// TIA Portal project "2022.10.20_FB_Auto-Hand视觉分拣急停" (V17)
// Vorlageprojekt für das Buch mit Zielsystem S7-1200

(* hardware
DEVICE "S7-1200-Station_1"  S7-1200 Station
   slot 0: "Baugruppenträger_0"  Rack  V1.0
   slot 1: "PLC_1"  CPU 1214C DC/DC/Rly  6ES7 214-1HG40-0XB0  V4.5
DEVICE "HMI_1"  KTP700 Basic PN
   slot 0: "HMI_1"  KTP700 Basic PN  6AV2 123-2GB03-0AX0  17.0.0.0
   slot 1: "HMI_RT_1"  KTP700 Basic PN  6AV2 123-2GB03-0AX0  17.0.0.0
   slot 5: "HMI_1.IE_CP_1"  PROFINET Interface  17.0.0.0
      slot 1: "PROFINET Interface_1"  PROFINET Interface
         slot 1: "Port_1"  Port
*)

// ===== PLC "PLC_1"  CPU 1214C DC/DC/Rly =====

VAR_GLOBAL   // PLC tag table "Standard-Variablentabelle"
   "复位按钮" AT %I0.2 : Bool;
   "System_Byte" AT %MB1 : Byte;
   "FirstScan" AT %M1.0 : Bool;
   "DiagStatusUpdate" AT %M1.1 : Bool;
   "AlwaysTRUE" AT %M1.2 : Bool;
   "AlwaysFALSE" AT %M1.3 : Bool;
   "Clock_Byte" AT %MB0 : Byte;
   "Clock_10Hz" AT %M0.0 : Bool;
   "Clock_5Hz" AT %M0.1 : Bool;
   "Clock_2.5Hz" AT %M0.2 : Bool;
   "Clock_2Hz" AT %M0.3 : Bool;
   "Clock_1.25Hz" AT %M0.4 : Bool;
   "Clock_1Hz" AT %M0.5 : Bool;
   "Clock_0.625Hz" AT %M0.6 : Bool;
   "Clock_0.5Hz" AT %M0.7 : Bool;
END_VAR

VAR_GLOBAL   // PLC tag table "XML 中的变量表_1"
   "启动按钮" AT %I0.0 : Bool;
   "停止按钮" AT %I0.1 : Bool;
   "复位信号" AT %Q0.2 : Bool;
   "急停" AT %I0.3 : Bool;
   "左电传感器" AT %I0.5 : Bool;
   "后电传感器" AT %I0.7 : Bool;
   "手动模式" AT %I1.0 : Bool;
   "自动模式" AT %I1.1 : Bool;
   "启动指示灯" AT %Q0.0 : Bool;
   "停止指示灯" AT %Q0.1 : Bool;
   "送料带" AT %Q0.3 : Bool;
   "直行电机" AT %Q0.4 : Bool;
   "左换向" AT %Q0.5 : Bool;
   "右换向" AT %Q0.6 : Bool;
   "后1带—原料" AT %Q0.7 : Bool;
   "右1带—基座" AT %Q1.0 : Bool;
   "左1带_产品盖" AT %Q1.1 : Bool;
   "出料台" AT %Q1.2 : Bool;
   "挡板" AT %Q1.3 : Bool;
   "视觉相机" AT %ID30 : DWord;
   "右电传感器" AT %I0.6 : Bool;
END_VAR

DATA_BLOCK "主程序DB"   // DB1
{ S7_Optimized_Access := 'TRUE' }
VERSION : 0.1
   VAR
      核心分拣区程序步 : Int;
      启动按钮 : Bool;
      停止按钮 : Bool;
      复位按钮 : Bool;
      急停按钮 : Bool := true;
      "手/自动切换" : Bool;
      中间变量1 : Bool;
      中间变量2 : Bool;
      中间变量3 : Bool;
      中间变量4 : Bool;
      中间变量5 : Bool;
      运行模式 : Int;
   END_VAR
BEGIN
END_DATA_BLOCK

// folder: 01核心分拣区

DATA_BLOCK "视觉核心分拣区FB块_DB"   // DB2
{ S7_Optimized_Access := 'TRUE' }
VERSION : 0.1
// stored: InstanceOfName 视觉核心分拣区FB块
"视觉核心分拣区FB块"
BEGIN
END_DATA_BLOCK

// folder: 02自动运行模式

DATA_BLOCK "自动运行_DB_1"   // DB7
{ S7_Optimized_Access := 'TRUE' }
VERSION : 0.1
// stored: InstanceOfName 自动运行
"自动运行"
BEGIN
END_DATA_BLOCK

// folder: 03手动运行模式

DATA_BLOCK "手动运行_DB"   // DB4
{ S7_Optimized_Access := 'TRUE' }
VERSION : 0.1
// stored: InstanceOfName 手动运行
"手动运行"
BEGIN
END_DATA_BLOCK

DATA_BLOCK "视觉核心分拣区FB块_DB_1"   // DB5
{ S7_Optimized_Access := 'TRUE' }
VERSION : 0.1
// stored: InstanceOfName 视觉核心分拣区FB块
"视觉核心分拣区FB块"
BEGIN
END_DATA_BLOCK

// folder: 系统急停

DATA_BLOCK "系统急停_DB"   // DB6
{ S7_Optimized_Access := 'TRUE' }
VERSION : 0.1
// stored: InstanceOfName 系统急停
"系统急停"
BEGIN
END_DATA_BLOCK

// folder: (top level)

FUNCTION "MHJ-PLC-Lab-Function-S71200" : Void   // FC9000, SCL
{ S7_Optimized_Access := 'TRUE' }
VERSION : 0.1
   VAR_TEMP
      rdTimeReturn : Int;
      outputTime : DTL;
      SyncVal : Byte;
      forVal : Int;
      forVal_2 : Int;
      Value : Byte;
   END_VAR
   VAR CONSTANT
      CompVal : Byte := 16#34;
      Value_01 : Byte := 16#11;
      Value_01_DW : DWord := 16#A165_D992;
      Value_02_DW : DWord := 16#58BE_4401;
   END_VAR
BEGIN

   #Value:=PEEK(area := 16#82,
        dbNumber := 0,
        byteOffset := 511);
   #Value := #Value + 1;

   POKE(area := 16#82,
        dbNumber := 0,
        byteOffset := 511,
        value := #Value);

   POKE(area:=16#81,
        dbNumber:=0,
        byteOffset:=1016,
        value:=#Value_01_DW);
   POKE(area := 16#81,
        dbNumber := 0,
        byteOffset := 1020,
        value := #Value_02_DW);

   POKE(area := 16#81,
        dbNumber := 0,
        byteOffset := 511,
        value := B#16#00);

   FOR #forVal := 0 TO 120 DO
       FOR #forVal_2:=0 TO 10 DO
           #rdTimeReturn:=RD_SYS_T(#outputTime);
           #rdTimeReturn := WR_SYS_T(#outputTime);
           #rdTimeReturn := RD_SYS_T(#outputTime);
           #rdTimeReturn := WR_SYS_T(#outputTime);
       END_FOR;
       #SyncVal:= PEEK(area := 16#81,
                      dbNumber := 0,
                      byteOffset := 511);
       IF #SyncVal = #CompVal THEN
          GOTO M_1;
       END_IF;
   END_FOR;
   RETURN;

   M_1:
   POKE(area := 16#81,
        dbNumber := 0,
        byteOffset := 511,
        value := B#16#0);
END_FUNCTION

ORGANIZATION_BLOCK "Main"   // OB1, LAD, ProgramCycle
TITLE = "Main Program Sweep (Cycle)"
{ S7_Optimized_Access := 'TRUE' }
VERSION : 0.1
   VAR_INPUT
      Initial_Call : Bool;   // Initial call of this OB
      Remanence : Bool;   // =True, if remanent data are available
   END_VAR
   VAR_TEMP   // added for the SCL form of the ladder/FBD networks
      _w1 : Bool;
      _w2 : Bool;
      _w3 : Bool;
   END_VAR
BEGIN

REGION Network 1: Konnektierungsbaustein für PLC-Lab
   // Im Netzwerk 1 wird der Konnektierungsbaustein für PLC-Lab aufgerufen.
   // Dieser Aufruf darf nicht entfernt werden!
   // Factory_调试按钮时，需要人工触发的一开始点开，亮成闪电状，需要触发的调成没有故障，白色小眼睛
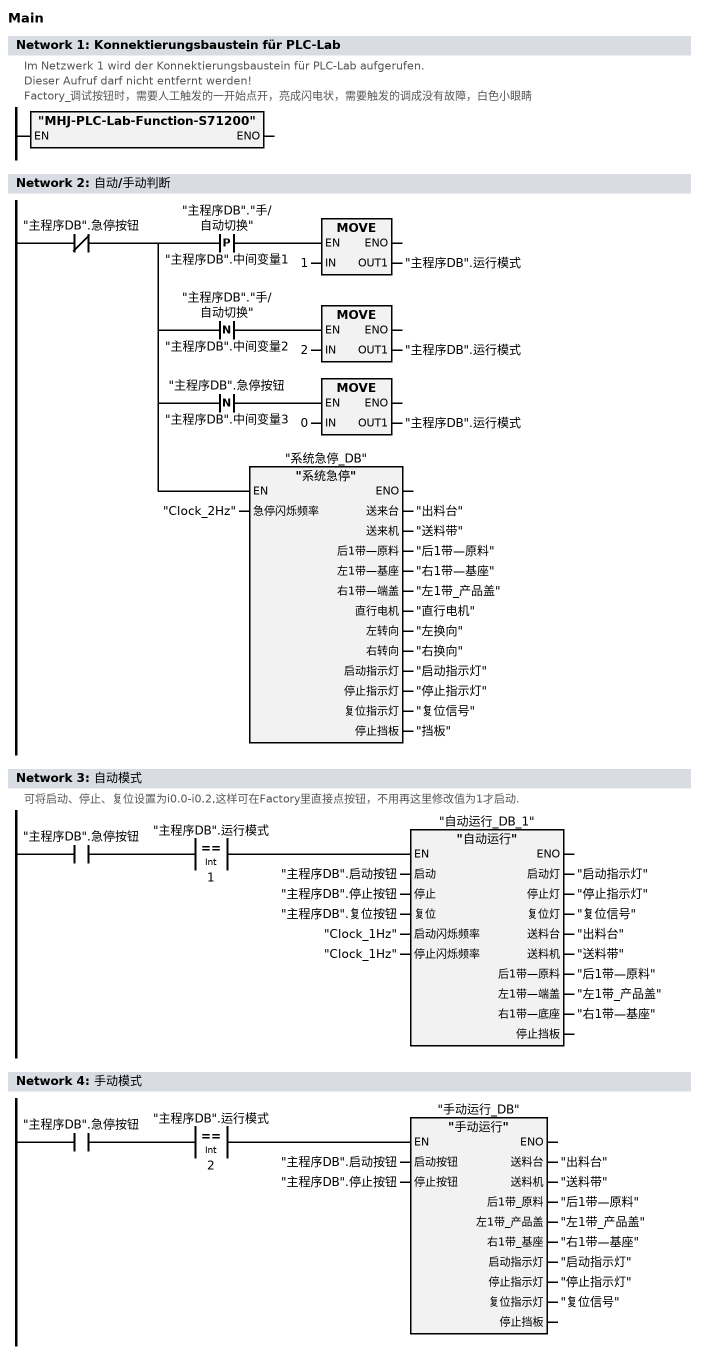
   RUNG wire#powerrail
      "MHJ-PLC-Lab-Function-S71200"()
   END_RUNG
   // the same network as SCL:
   "MHJ-PLC-Lab-Function-S71200"();
END_REGION

REGION Network 2: 自动/手动判断
   RUNG wire#powerrail
      I_Contact( "主程序DB".急停按钮 )
      wire#w1
      P_Contact(operand := "主程序DB"."手/自动切换", bit := "主程序DB".中间变量1)
      Move(in := 1, out1 => "主程序DB".运行模式)
   END_RUNG
   RUNG wire#w1
      N_Contact(operand := "主程序DB"."手/自动切换", bit := "主程序DB".中间变量2)
      Move(in := 2, out1 => "主程序DB".运行模式)
   END_RUNG
   RUNG wire#w1
      N_Contact(operand := "主程序DB".急停按钮, bit := "主程序DB".中间变量3)
      Move(in := 0, out1 => "主程序DB".运行模式)
   END_RUNG
   RUNG wire#w1
      "系统急停_DB"(急停闪烁频率 := "Clock_2Hz", 送来台 => "出料台", 送来机 => "送料带", "后1带—原料" => "后1带—原料", "左1带—基座" => "右1带—基座", "右1带—端盖" => "左1带_产品盖", 直行电机 => "直行电机", 左转向 => "左换向", 右转向 => "右换向", 启动指示灯 => "启动指示灯", 停止指示灯 => "停止指示灯", 复位指示灯 => "复位信号", 停止挡板 => "挡板")
   END_RUNG
   // the same network as SCL:
   #_w1 := NOT "主程序DB".急停按钮 AND "主程序DB"."手/自动切换" AND NOT "主程序DB".中间变量1;   // rising edge of "主程序DB"."手/自动切换"
   "主程序DB".中间变量1 := "主程序DB"."手/自动切换";
   IF #_w1 THEN "主程序DB".运行模式 := 1; END_IF;
   #_w2 := NOT "主程序DB".急停按钮 AND NOT "主程序DB"."手/自动切换" AND "主程序DB".中间变量2;   // falling edge of "主程序DB"."手/自动切换"
   "主程序DB".中间变量2 := "主程序DB"."手/自动切换";
   IF #_w2 THEN "主程序DB".运行模式 := 2; END_IF;
   #_w3 := NOT "主程序DB".急停按钮 AND NOT "主程序DB".急停按钮 AND "主程序DB".中间变量3;   // falling edge of "主程序DB".急停按钮
   "主程序DB".中间变量3 := "主程序DB".急停按钮;
   IF #_w3 THEN "主程序DB".运行模式 := 0; END_IF;
   IF NOT "主程序DB".急停按钮 THEN
       "系统急停_DB"(急停闪烁频率 := "Clock_2Hz",   // "系统急停"
                 送来台 => "出料台",
                 送来机 => "送料带",
                 "后1带—原料" => "后1带—原料",
                 "左1带—基座" => "右1带—基座",
                 "右1带—端盖" => "左1带_产品盖",
                 直行电机 => "直行电机",
                 左转向 => "左换向",
                 右转向 => "右换向",
                 启动指示灯 => "启动指示灯",
                 停止指示灯 => "停止指示灯",
                 复位指示灯 => "复位信号",
                 停止挡板 => "挡板");
   END_IF;
END_REGION

REGION Network 3: 自动模式
   // 可将启动、停止、复位设置为i0.0-i0.2,这样可在Factory里直接点按钮，不用再这里修改值为1才启动.
   RUNG wire#powerrail
      Contact( "主程序DB".急停按钮 )
      { S7_Templates := "SrcType := Int" } EQ_Contact(in1 := "主程序DB".运行模式, in2 := 1)
      "自动运行_DB_1"(启动 := "主程序DB".启动按钮, 停止 := "主程序DB".停止按钮, 复位 := "主程序DB".复位按钮, 启动闪烁频率 := "Clock_1Hz", 停止闪烁频率 := "Clock_1Hz", 启动灯 => "启动指示灯", 停止灯 => "停止指示灯", 复位灯 => "复位信号", 送料台 => "出料台", 送料机 => "送料带", "后1带—原料" => "后1带—原料", "左1带—端盖" => "左1带_产品盖", "右1带—底座" => "右1带—基座", 停止挡板 =>)
   END_RUNG
   // the same network as SCL:
   IF "主程序DB".急停按钮 AND ("主程序DB".运行模式 = 1) THEN
       "自动运行_DB_1"(启动 := "主程序DB".启动按钮,   // "自动运行"
                   停止 := "主程序DB".停止按钮,
                   复位 := "主程序DB".复位按钮,
                   启动闪烁频率 := "Clock_1Hz",
                   停止闪烁频率 := "Clock_1Hz",
                   启动灯 => "启动指示灯",
                   停止灯 => "停止指示灯",
                   复位灯 => "复位信号",
                   送料台 => "出料台",
                   送料机 => "送料带",
                   "后1带—原料" => "后1带—原料",
                   "左1带—端盖" => "左1带_产品盖",
                   "右1带—底座" => "右1带—基座");
   END_IF;
END_REGION

REGION Network 4: 手动模式
   RUNG wire#powerrail
      Contact( "主程序DB".急停按钮 )
      { S7_Templates := "SrcType := Int" } EQ_Contact(in1 := "主程序DB".运行模式, in2 := 2)
      "手动运行_DB"(启动按钮 := "主程序DB".启动按钮, 停止按钮 := "主程序DB".停止按钮, 送料台 => "出料台", 送料机 => "送料带", 后1带_原料 => "后1带—原料", 左1带_产品盖 => "左1带_产品盖", 右1带_基座 => "右1带—基座", 启动指示灯 => "启动指示灯", 停止指示灯 => "停止指示灯", 复位指示灯 => "复位信号", 停止挡板 =>)
   END_RUNG
   // the same network as SCL:
   IF "主程序DB".急停按钮 AND ("主程序DB".运行模式 = 2) THEN
       "手动运行_DB"(启动按钮 := "主程序DB".启动按钮,   // "手动运行"
                 停止按钮 := "主程序DB".停止按钮,
                 送料台 => "出料台",
                 送料机 => "送料带",
                 后1带_原料 => "后1带—原料",
                 左1带_产品盖 => "左1带_产品盖",
                 右1带_基座 => "右1带—基座",
                 启动指示灯 => "启动指示灯",
                 停止指示灯 => "停止指示灯",
                 复位指示灯 => "复位信号");
   END_IF;
END_REGION
END_ORGANIZATION_BLOCK

// folder: 01核心分拣区

FUNCTION_BLOCK "视觉核心分拣区FB块"   // FB1, LAD
{ S7_Optimized_Access := 'TRUE' }
VERSION : 0.1
   VAR_INPUT
      视觉相机数据 : DWord;
      后电传感器 : Bool;
      左电传感器 : Bool;
      右电传感器 : Bool;
   END_VAR
   VAR_OUTPUT
      直行电机 : Bool;
      左转向 : Bool;
      右转向 : Bool;
   END_VAR
   VAR_IN_OUT
      程序步 : Int;
   END_VAR
   VAR
      中间变量1 : Bool;
      中间变量2 : Bool;
      中间变量3 : Bool;
   END_VAR
   VAR_TEMP   // added for the SCL form of the ladder/FBD networks
      _w1 : Bool;
   END_VAR
BEGIN

REGION Network 1: 物料判断
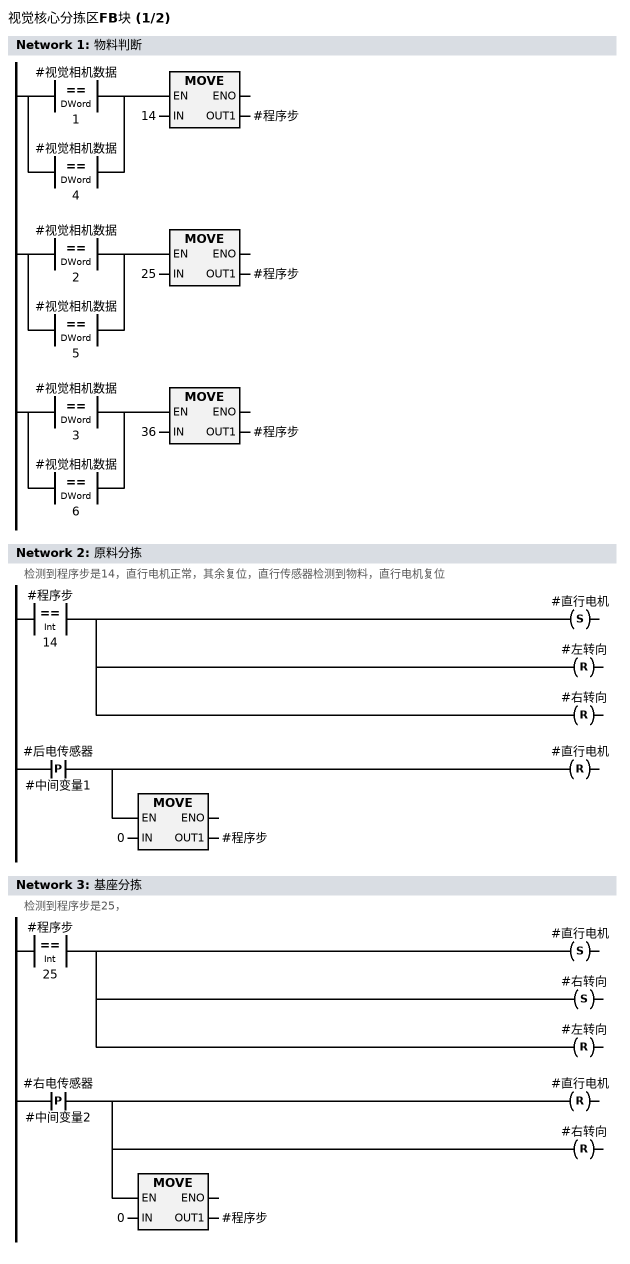
   RUNG wire#powerrail
      { S7_Templates := "SrcType := DWord" } EQ_Contact(in1 := #视觉相机数据, in2 := 1)
      wire#w1
      Move(in := 14, out1 => #程序步)
   END_RUNG
   RUNG wire#powerrail
      { S7_Templates := "SrcType := DWord" } EQ_Contact(in1 := #视觉相机数据, in2 := 4)
   END_RUNG wire#w1
   RUNG wire#powerrail
      { S7_Templates := "SrcType := DWord" } EQ_Contact(in1 := #视觉相机数据, in2 := 2)
      wire#w2
      Move(in := 25, out1 => #程序步)
   END_RUNG
   RUNG wire#powerrail
      { S7_Templates := "SrcType := DWord" } EQ_Contact(in1 := #视觉相机数据, in2 := 5)
   END_RUNG wire#w2
   RUNG wire#powerrail
      { S7_Templates := "SrcType := DWord" } EQ_Contact(in1 := #视觉相机数据, in2 := 3)
      wire#w3
      Move(in := 36, out1 => #程序步)
   END_RUNG
   RUNG wire#powerrail
      { S7_Templates := "SrcType := DWord" } EQ_Contact(in1 := #视觉相机数据, in2 := 6)
   END_RUNG wire#w3
   // the same network as SCL:
   IF (#视觉相机数据 = 1) OR (#视觉相机数据 = 4) THEN #程序步 := 14; END_IF;
   IF (#视觉相机数据 = 2) OR (#视觉相机数据 = 5) THEN #程序步 := 25; END_IF;
   IF (#视觉相机数据 = 3) OR (#视觉相机数据 = 6) THEN #程序步 := 36; END_IF;
END_REGION

REGION Network 2: 原料分拣
   // 检测到程序步是14，直行电机正常，其余复位，直行传感器检测到物料，直行电机复位
   RUNG wire#powerrail
      { S7_Templates := "SrcType := Int" } EQ_Contact(in1 := #程序步, in2 := 14)
      wire#w1
      S_Coil( #直行电机 )
   END_RUNG
   RUNG wire#w1
      R_Coil( #左转向 )
   END_RUNG
   RUNG wire#w1
      R_Coil( #右转向 )
   END_RUNG
   RUNG wire#powerrail
      P_Contact(operand := #后电传感器, bit := #中间变量1)
      wire#w2
      R_Coil( #直行电机 )
   END_RUNG
   RUNG wire#w2
      Move(in := 0, out1 => #程序步)
   END_RUNG
   // the same network as SCL:
   IF #程序步 = 14 THEN
       #直行电机 := TRUE;
       #左转向 := FALSE;
       #右转向 := FALSE;
   END_IF;
   #_w1 := #后电传感器 AND NOT #中间变量1;   // rising edge of #后电传感器
   #中间变量1 := #后电传感器;
   IF #_w1 THEN
       #直行电机 := FALSE;
       #程序步 := 0;
   END_IF;
END_REGION

REGION Network 3: 基座分拣
   // 检测到程序步是25，
   RUNG wire#powerrail
      { S7_Templates := "SrcType := Int" } EQ_Contact(in1 := #程序步, in2 := 25)
      wire#w1
      S_Coil( #直行电机 )
   END_RUNG
   RUNG wire#w1
      S_Coil( #右转向 )
   END_RUNG
   RUNG wire#w1
      R_Coil( #左转向 )
   END_RUNG
   RUNG wire#powerrail
      P_Contact(operand := #右电传感器, bit := #中间变量2)
      wire#w2
      R_Coil( #直行电机 )
   END_RUNG
   RUNG wire#w2
      R_Coil( #右转向 )
   END_RUNG
   RUNG wire#w2
      Move(in := 0, out1 => #程序步)
   END_RUNG
   // the same network as SCL:
   IF #程序步 = 25 THEN
       #直行电机 := TRUE;
       #右转向 := TRUE;
       #左转向 := FALSE;
   END_IF;
   #_w1 := #右电传感器 AND NOT #中间变量2;   // rising edge of #右电传感器
   #中间变量2 := #右电传感器;
   IF #_w1 THEN
       #直行电机 := FALSE;
       #右转向 := FALSE;
       #程序步 := 0;
   END_IF;
END_REGION

REGION Network 4: 基盖
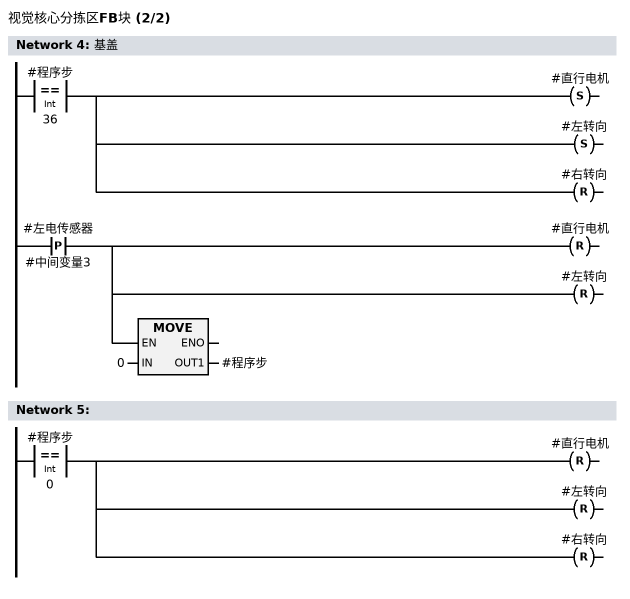
   RUNG wire#powerrail
      { S7_Templates := "SrcType := Int" } EQ_Contact(in1 := #程序步, in2 := 36)
      wire#w1
      S_Coil( #直行电机 )
   END_RUNG
   RUNG wire#w1
      S_Coil( #左转向 )
   END_RUNG
   RUNG wire#w1
      R_Coil( #右转向 )
   END_RUNG
   RUNG wire#powerrail
      P_Contact(operand := #左电传感器, bit := #中间变量3)
      wire#w2
      R_Coil( #直行电机 )
   END_RUNG
   RUNG wire#w2
      R_Coil( #左转向 )
   END_RUNG
   RUNG wire#w2
      Move(in := 0, out1 => #程序步)
   END_RUNG
   // the same network as SCL:
   IF #程序步 = 36 THEN
       #直行电机 := TRUE;
       #左转向 := TRUE;
       #右转向 := FALSE;
   END_IF;
   #_w1 := #左电传感器 AND NOT #中间变量3;   // rising edge of #左电传感器
   #中间变量3 := #左电传感器;
   IF #_w1 THEN
       #直行电机 := FALSE;
       #左转向 := FALSE;
       #程序步 := 0;
   END_IF;
END_REGION

REGION Network 5
   RUNG wire#powerrail
      { S7_Templates := "SrcType := Int" } EQ_Contact(in1 := #程序步, in2 := 0)
      wire#w1
      R_Coil( #直行电机 )
   END_RUNG
   RUNG wire#w1
      R_Coil( #左转向 )
   END_RUNG
   RUNG wire#w1
      R_Coil( #右转向 )
   END_RUNG
   // the same network as SCL:
   IF #程序步 = 0 THEN
       #直行电机 := FALSE;
       #左转向 := FALSE;
       #右转向 := FALSE;
   END_IF;
END_REGION
END_FUNCTION_BLOCK

// folder: 02自动运行模式

FUNCTION_BLOCK "自动运行"   // FB2, LAD
{ S7_Optimized_Access := 'TRUE' }
VERSION : 0.1
   VAR_INPUT
      启动 : Bool;
      停止 : Bool;
      复位 : Bool;
      启动闪烁频率 : Bool;
      停止闪烁频率 : Bool;
   END_VAR
   VAR_OUTPUT
      启动灯 : Bool;
      停止灯 : Bool;
      复位灯 : Bool;
      送料台 : Bool;
      送料机 : Bool;
      "后1带—原料" : Bool;
      "左1带—端盖" : Bool;
      "右1带—底座" : Bool;
      停止挡板 : Bool;
   END_VAR
   VAR
      自动运行启动中 : Bool;
      自动运行启动完成 : Bool;
      自动停止进行中 : Bool;
      自动停止完成 : Bool;
      中间变量1 : Bool;
      中间变量2 : Bool;
      中间变量3 : Bool;
      中间变量4 : Bool;
      中间变量5 : Bool;
      中间变量6 : Bool;
      中间变量7 : Bool;
      IEC_Timer_0_Instance_01 : TON_TIME;
      IEC_Timer_0_Instance_02 : TON_TIME;
   END_VAR
   VAR_TEMP   // added for the SCL form of the ladder/FBD networks
      _w1 : Bool;
      _w2 : Bool;
   END_VAR
BEGIN

REGION Network 1: 启动二级输送机
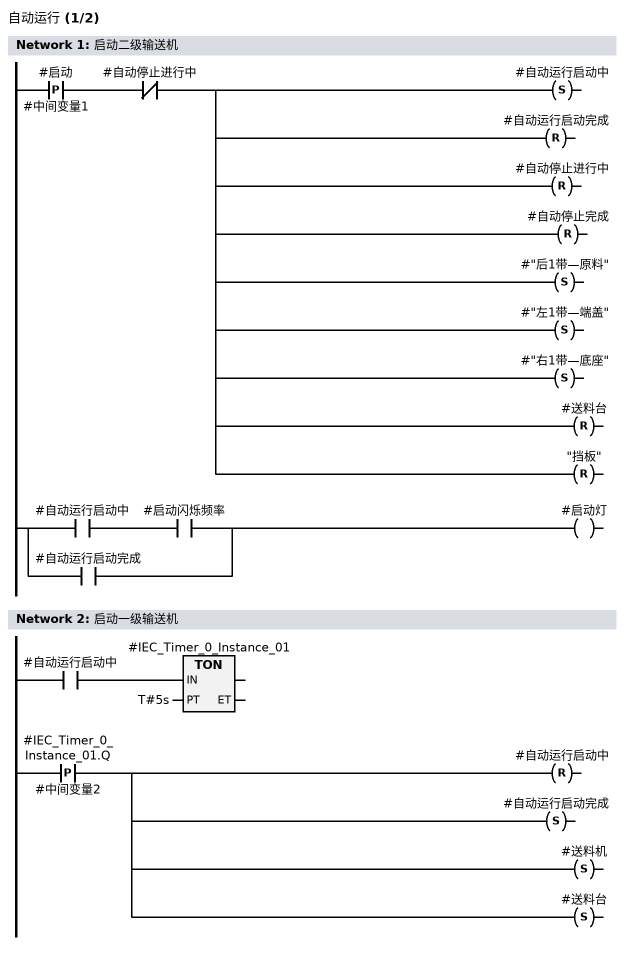
   RUNG wire#powerrail
      P_Contact(operand := #启动, bit := #中间变量1)
      I_Contact( #自动停止进行中 )
      wire#w1
      S_Coil( #自动运行启动中 )
   END_RUNG
   RUNG wire#w1
      R_Coil( #自动运行启动完成 )
   END_RUNG
   RUNG wire#w1
      R_Coil( #自动停止进行中 )
   END_RUNG
   RUNG wire#w1
      R_Coil( #自动停止完成 )
   END_RUNG
   RUNG wire#w1
      S_Coil( #"后1带—原料" )
   END_RUNG
   RUNG wire#w1
      S_Coil( #"左1带—端盖" )
   END_RUNG
   RUNG wire#w1
      S_Coil( #"右1带—底座" )
   END_RUNG
   RUNG wire#w1
      R_Coil( #送料台 )
   END_RUNG
   RUNG wire#w1
      R_Coil( "挡板" )
   END_RUNG
   RUNG wire#powerrail
      Contact( #自动运行启动中 )
      Contact( #启动闪烁频率 )
      wire#w2
      Coil( #启动灯 )
   END_RUNG
   RUNG wire#powerrail
      Contact( #自动运行启动完成 )
   END_RUNG wire#w2
   // the same network as SCL:
   #_w1 := #启动 AND NOT #中间变量1;   // rising edge of #启动
   #中间变量1 := #启动;
   IF #_w1 AND NOT #自动停止进行中 THEN
       #自动运行启动中 := TRUE;
       #自动运行启动完成 := FALSE;
   END_IF;
   #_w2 := #_w1 AND NOT #自动停止进行中;
   IF #_w2 THEN
       #自动停止进行中 := FALSE;
       #自动停止完成 := FALSE;
       #"后1带—原料" := TRUE;
       #"左1带—端盖" := TRUE;
       #"右1带—底座" := TRUE;
       #送料台 := FALSE;
       "挡板" := FALSE;
   END_IF;
   #启动灯 := (#自动运行启动中 AND #启动闪烁频率) OR #自动运行启动完成;
END_REGION

REGION Network 2: 启动一级输送机
   #IEC_Timer_0_Instance_01(IN := #自动运行启动中, PT := T#5s);   // TON
   #_w1 := #IEC_Timer_0_Instance_01.Q AND NOT #中间变量2;   // rising edge of #IEC_Timer_0_Instance_01.Q
   #中间变量2 := #IEC_Timer_0_Instance_01.Q;
   IF #_w1 THEN
       #自动运行启动中 := FALSE;
       #自动运行启动完成 := TRUE;
       #送料机 := TRUE;
       #送料台 := TRUE;
   END_IF;
END_REGION

REGION Network 3: 一级输送机停止运行
   // 加入自动运行启动中，是为防止启动时，按下停止按钮,两者同时运行出现bug。
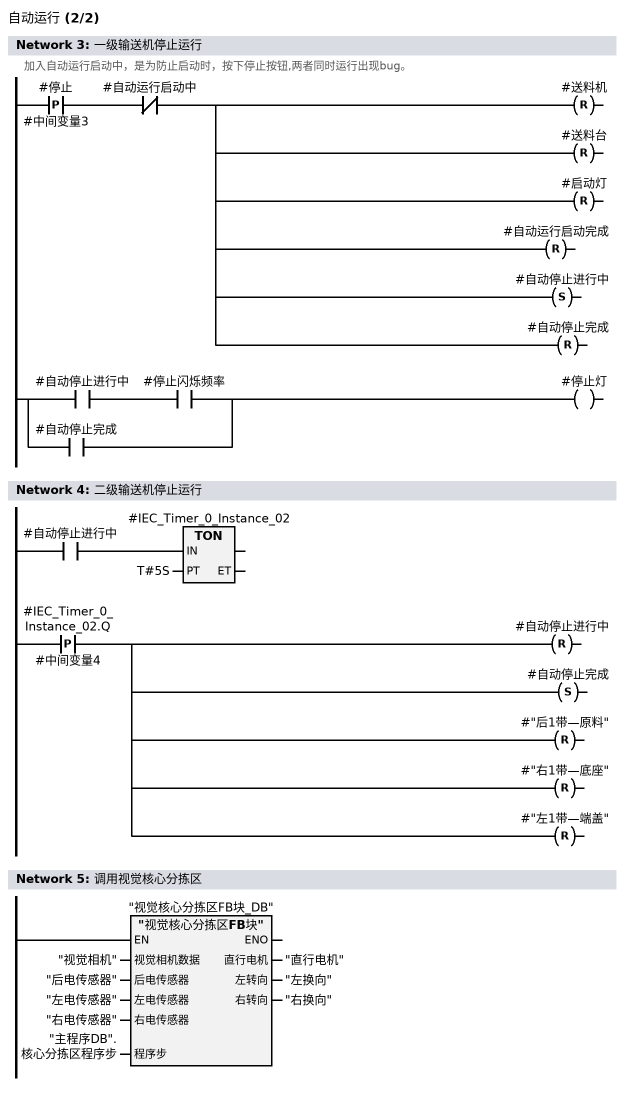
   RUNG wire#powerrail
      P_Contact(operand := #停止, bit := #中间变量3)
      I_Contact( #自动运行启动中 )
      wire#w1
      R_Coil( #送料机 )
   END_RUNG
   RUNG wire#w1
      R_Coil( #送料台 )
   END_RUNG
   RUNG wire#w1
      R_Coil( #启动灯 )
   END_RUNG
   RUNG wire#w1
      R_Coil( #自动运行启动完成 )
   END_RUNG
   RUNG wire#w1
      S_Coil( #自动停止进行中 )
   END_RUNG
   RUNG wire#w1
      R_Coil( #自动停止完成 )
   END_RUNG
   RUNG wire#powerrail
      Contact( #自动停止进行中 )
      Contact( #停止闪烁频率 )
      wire#w2
      Coil( #停止灯 )
   END_RUNG
   RUNG wire#powerrail
      Contact( #自动停止完成 )
   END_RUNG wire#w2
   // the same network as SCL:
   #_w1 := #停止 AND NOT #中间变量3;   // rising edge of #停止
   #中间变量3 := #停止;
   IF #_w1 AND NOT #自动运行启动中 THEN
       #送料机 := FALSE;
       #送料台 := FALSE;
       #启动灯 := FALSE;
       #自动运行启动完成 := FALSE;
       #自动停止进行中 := TRUE;
       #自动停止完成 := FALSE;
   END_IF;
   #停止灯 := (#自动停止进行中 AND #停止闪烁频率) OR #自动停止完成;
END_REGION

REGION Network 4: 二级输送机停止运行
   #IEC_Timer_0_Instance_02(IN := #自动停止进行中, PT := T#5S);   // TON
   #_w1 := #IEC_Timer_0_Instance_02.Q AND NOT #中间变量4;   // rising edge of #IEC_Timer_0_Instance_02.Q
   #中间变量4 := #IEC_Timer_0_Instance_02.Q;
   IF #_w1 THEN
       #自动停止进行中 := FALSE;
       #自动停止完成 := TRUE;
       #"后1带—原料" := FALSE;
       #"右1带—底座" := FALSE;
       #"左1带—端盖" := FALSE;
   END_IF;
END_REGION

REGION Network 5: 调用视觉核心分拣区
   RUNG wire#powerrail
      "视觉核心分拣区FB块_DB"(视觉相机数据 := "视觉相机", 后电传感器 := "后电传感器", 左电传感器 := "左电传感器", 右电传感器 := "右电传感器", 程序步 := "主程序DB".核心分拣区程序步, 直行电机 => "直行电机", 左转向 => "左换向", 右转向 => "右换向")
   END_RUNG
   // the same network as SCL:
   "视觉核心分拣区FB块_DB"(视觉相机数据 := "视觉相机",   // "视觉核心分拣区FB块"
                   后电传感器 := "后电传感器",
                   左电传感器 := "左电传感器",
                   右电传感器 := "右电传感器",
                   程序步 := "主程序DB".核心分拣区程序步,
                   直行电机 => "直行电机",
                   左转向 => "左换向",
                   右转向 => "右换向");
END_REGION
END_FUNCTION_BLOCK

// folder: 03手动运行模式

FUNCTION_BLOCK "手动运行"   // FB3, LAD
{ S7_Optimized_Access := 'TRUE' }
VERSION : 0.1
   VAR_INPUT
      启动按钮 : Bool;
      停止按钮 : Bool;
   END_VAR
   VAR_OUTPUT
      送料台 : Bool;
      送料机 : Bool;
      后1带_原料 : Bool;
      左1带_产品盖 : Bool;
      右1带_基座 : Bool;
      启动指示灯 : Bool;
      停止指示灯 : Bool;
      复位指示灯 : Bool;
      停止挡板 : Bool;
   END_VAR
   VAR
      中间标志位1 : Bool;
      中间标志位2 : Bool;
      中间标志位3 : Bool;
      中间标志位4 : Bool;
      中间标志位5 : Bool;
   END_VAR
   VAR_TEMP   // added for the SCL form of the ladder/FBD networks
      _w1 : Bool;
   END_VAR
BEGIN

REGION Network 1: 启动
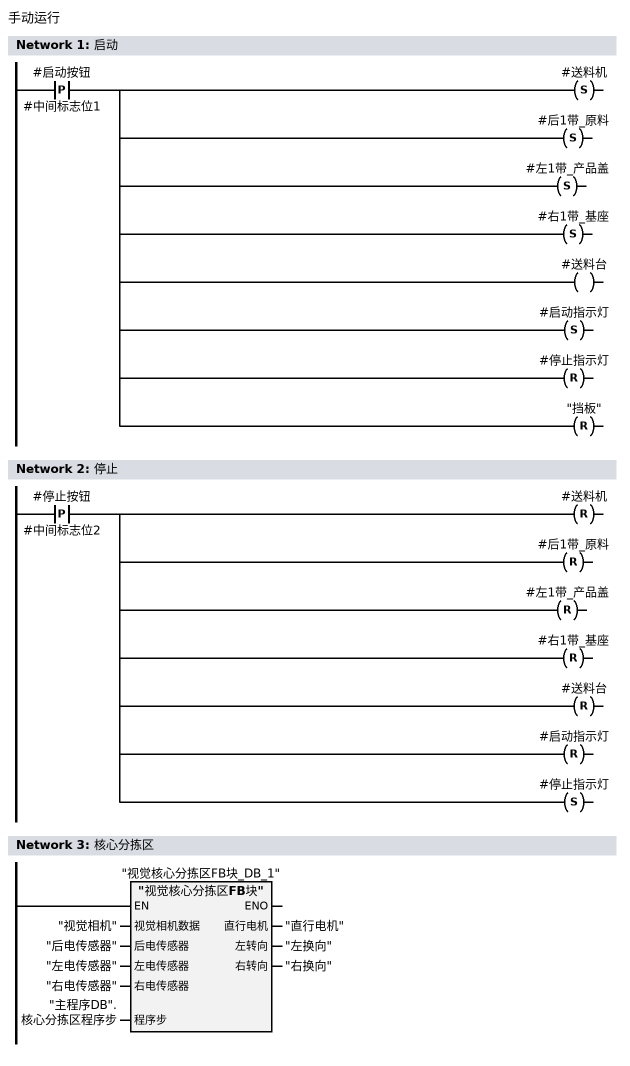
   RUNG wire#powerrail
      P_Contact(operand := #启动按钮, bit := #中间标志位1)
      wire#w1
      S_Coil( #送料机 )
   END_RUNG
   RUNG wire#w1
      S_Coil( #后1带_原料 )
   END_RUNG
   RUNG wire#w1
      S_Coil( #左1带_产品盖 )
   END_RUNG
   RUNG wire#w1
      S_Coil( #右1带_基座 )
   END_RUNG
   RUNG wire#w1
      Coil( #送料台 )
   END_RUNG
   RUNG wire#w1
      S_Coil( #启动指示灯 )
   END_RUNG
   RUNG wire#w1
      R_Coil( #停止指示灯 )
   END_RUNG
   RUNG wire#w1
      R_Coil( "挡板" )
   END_RUNG
   // the same network as SCL:
   #_w1 := #启动按钮 AND NOT #中间标志位1;   // rising edge of #启动按钮
   #中间标志位1 := #启动按钮;
   IF #_w1 THEN
       #送料机 := TRUE;
       #后1带_原料 := TRUE;
       #左1带_产品盖 := TRUE;
       #右1带_基座 := TRUE;
   END_IF;
   #送料台 := #_w1;
   IF #_w1 THEN
       #启动指示灯 := TRUE;
       #停止指示灯 := FALSE;
       "挡板" := FALSE;
   END_IF;
END_REGION

REGION Network 2: 停止
   RUNG wire#powerrail
      P_Contact(operand := #停止按钮, bit := #中间标志位2)
      wire#w1
      R_Coil( #送料机 )
   END_RUNG
   RUNG wire#w1
      R_Coil( #后1带_原料 )
   END_RUNG
   RUNG wire#w1
      R_Coil( #左1带_产品盖 )
   END_RUNG
   RUNG wire#w1
      R_Coil( #右1带_基座 )
   END_RUNG
   RUNG wire#w1
      R_Coil( #送料台 )
   END_RUNG
   RUNG wire#w1
      R_Coil( #启动指示灯 )
   END_RUNG
   RUNG wire#w1
      S_Coil( #停止指示灯 )
   END_RUNG
   // the same network as SCL:
   #_w1 := #停止按钮 AND NOT #中间标志位2;   // rising edge of #停止按钮
   #中间标志位2 := #停止按钮;
   IF #_w1 THEN
       #送料机 := FALSE;
       #后1带_原料 := FALSE;
       #左1带_产品盖 := FALSE;
       #右1带_基座 := FALSE;
       #送料台 := FALSE;
       #启动指示灯 := FALSE;
       #停止指示灯 := TRUE;
   END_IF;
END_REGION

REGION Network 3: 核心分拣区
   RUNG wire#powerrail
      "视觉核心分拣区FB块_DB_1"(视觉相机数据 := "视觉相机", 后电传感器 := "后电传感器", 左电传感器 := "左电传感器", 右电传感器 := "右电传感器", 程序步 := "主程序DB".核心分拣区程序步, 直行电机 => "直行电机", 左转向 => "左换向", 右转向 => "右换向")
   END_RUNG
   // the same network as SCL:
   "视觉核心分拣区FB块_DB_1"(视觉相机数据 := "视觉相机",   // "视觉核心分拣区FB块"
                     后电传感器 := "后电传感器",
                     左电传感器 := "左电传感器",
                     右电传感器 := "右电传感器",
                     程序步 := "主程序DB".核心分拣区程序步,
                     直行电机 => "直行电机",
                     左转向 => "左换向",
                     右转向 => "右换向");
END_REGION
END_FUNCTION_BLOCK

// folder: 系统急停

FUNCTION_BLOCK "系统急停"   // FB4, LAD
{ S7_Optimized_Access := 'TRUE' }
VERSION : 0.1
   VAR_INPUT
      急停闪烁频率 : Bool;
   END_VAR
   VAR_OUTPUT
      送来台 : Bool;
      送来机 : Bool;
      "后1带—原料" : Bool;
      "左1带—基座" : Bool;
      "右1带—端盖" : Bool;
      直行电机 : Bool;
      左转向 : Bool;
      右转向 : Bool;
      启动指示灯 : Bool;
      停止指示灯 : Bool;
      复位指示灯 : Bool;
      停止挡板 : Bool;
   END_VAR
BEGIN

REGION Network 1
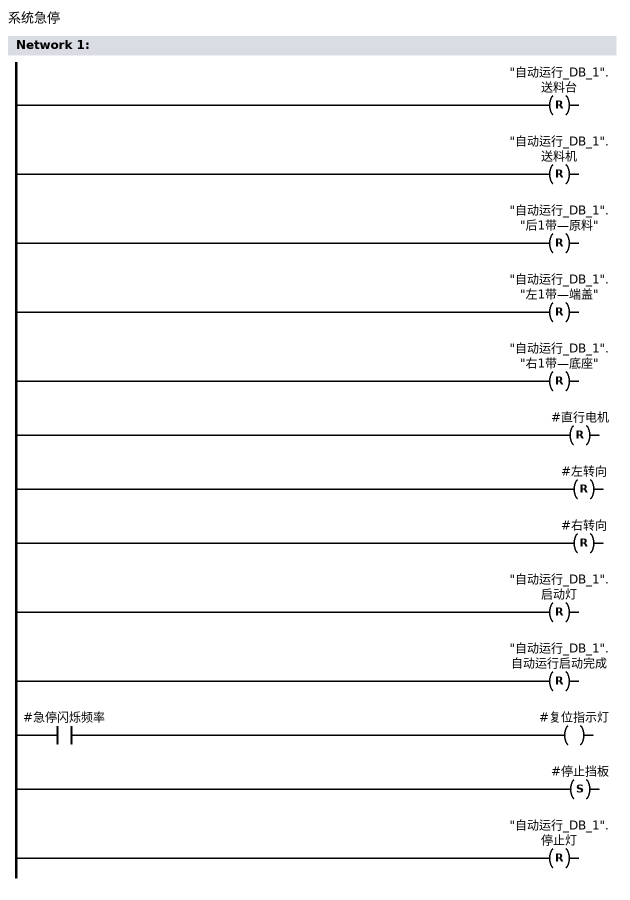
   RUNG wire#powerrail
      R_Coil( "自动运行_DB_1".送料台 )
   END_RUNG
   RUNG wire#powerrail
      R_Coil( "自动运行_DB_1".送料机 )
   END_RUNG
   RUNG wire#powerrail
      R_Coil( "自动运行_DB_1"."后1带—原料" )
   END_RUNG
   RUNG wire#powerrail
      R_Coil( "自动运行_DB_1"."左1带—端盖" )
   END_RUNG
   RUNG wire#powerrail
      R_Coil( "自动运行_DB_1"."右1带—底座" )
   END_RUNG
   RUNG wire#powerrail
      R_Coil( #直行电机 )
   END_RUNG
   RUNG wire#powerrail
      R_Coil( #左转向 )
   END_RUNG
   RUNG wire#powerrail
      R_Coil( #右转向 )
   END_RUNG
   RUNG wire#powerrail
      R_Coil( "自动运行_DB_1".启动灯 )
   END_RUNG
   RUNG wire#powerrail
      R_Coil( "自动运行_DB_1".自动运行启动完成 )
   END_RUNG
   RUNG wire#powerrail
      Contact( #急停闪烁频率 )
      Coil( #复位指示灯 )
   END_RUNG
   RUNG wire#powerrail
      S_Coil( #停止挡板 )
   END_RUNG
   RUNG wire#powerrail
      R_Coil( "自动运行_DB_1".停止灯 )
   END_RUNG
   // the same network as SCL:
   "自动运行_DB_1".送料台 := FALSE;
   "自动运行_DB_1".送料机 := FALSE;
   "自动运行_DB_1"."后1带—原料" := FALSE;
   "自动运行_DB_1"."左1带—端盖" := FALSE;
   "自动运行_DB_1"."右1带—底座" := FALSE;
   #直行电机 := FALSE;
   #左转向 := FALSE;
   #右转向 := FALSE;
   "自动运行_DB_1".启动灯 := FALSE;
   "自动运行_DB_1".自动运行启动完成 := FALSE;
   #复位指示灯 := #急停闪烁频率;
   #停止挡板 := TRUE;
   "自动运行_DB_1".停止灯 := FALSE;
END_REGION
END_FUNCTION_BLOCK

(* ===== HMI "HMI_RT_1" =====
system functions are stored by id; their names below are inferred from use
connection "HMI_连接_1": ETHERNET, SMART_S7_1200_OMS

HMI tags "默认变量表"
   "Tag_ScreenNumber" : UInt, internal
   "主程序DB_手/自动切换" : Bool = PLC 主程序DB.手/自动切换, 1 s
   "主程序DB_急停按钮" : Bool = PLC 主程序DB.急停按钮, 1 s
   "主程序DB_启动按钮" : Bool = PLC 主程序DB.启动按钮, 1 s
   "主程序DB_停止按钮" : Bool = PLC 主程序DB.停止按钮, 1 s
   "主程序DB_复位按钮" : Bool = PLC 主程序DB.复位按钮, 1 s

Template "模板_1" 800x480
   Button "Exit" at 714,429 size 71x50; TextOff 'Exit'; PictureOff "ExitRuntime_KTP700_Basic_PN_TR"; PictureOn "ExitRuntime_KTP700_Basic_PN_TR"
      on Release: StopRuntime(0)
   Button "Template_Button" at 614,429 size 71x50; TextOff 'Text'
   Button "Template_Button_1" at 514,429 size 71x50; TextOff 'Text'
   Button "Template_Button_2" at 414,429 size 71x50; TextOff 'Text'
   Button "Template_Button_3" at 314,429 size 71x50; TextOff 'Text'
   Button "Template_Button_4" at 214,429 size 71x50; TextOff 'Text'
   Button "Template_Button_5" at 114,429 size 71x50; TextOff 'Text'
   Button "Start screen" at 14,429 size 71x50; TextOff 'Start screen'; PictureOff "NavigateHome_KTP700_Basic_PN_TR"; PictureOn "NavigateHome_KTP700_Basic_PN_TR"
      on Release: ActivateScreen("根画面", 0)
   SymbolicIOField "Symbolic_IO_Field_Screen" at 93,9 size 600x33; TextOff '0'; TextOn '1'; TextList "TextList_ScreenNames"
      ProcessValue <- "Tag_ScreenNumber"
      on Change: ActivateScreenByNumber("Tag_ScreenNumber", 0)
   DateTimeField "HmiScreenItemData" at 695,25 size 105x25
   DateTimeField "HmiScreenItemData_1" at 695,0 size 105x25
   GraphicView "Logo" at 0,0 size 91x51; Picture "Logo of HMI_1"

screen "根画面" 800x480, template "模板_1"
   on GenerateScreen: SetTag("Tag_ScreenNumber", 1)
   Switch "开关_1" at 230,125 size 99x44; CaptionText 'Switch'; TextOff '手动'; TextOn '自动'
      ProcessValue <- "主程序DB_手/自动切换"
   Button "按钮_1" at 233,202 size 96x32; TextOff '急停'
      on Click: InvertBit("主程序DB_急停按钮")
   Button "按钮_2" at 501,131 size 96x32; TextOff '启动'
      on Press: SetBit("主程序DB_启动按钮")
      on Release: ResetBit("主程序DB_启动按钮")
   Button "按钮_3" at 504,192 size 96x32; TextOff '停止'
      on Press: SetBit("主程序DB_停止按钮")
      on Release: ResetBit("主程序DB_停止按钮")
   Button "按钮_4" at 503,250 size 96x32; TextOff '复位'
      on Press: SetBit("主程序DB_复位按钮")
      on Release: ResetBit("主程序DB_复位按钮")
   TextField "文本域_1" at 342,54 size 164x43; Text '视 觉 分 拣'
*)